PROGRAM MAIN
VAR
END_VAR

END_PROGRAM

(* stored: Version 1.1.0.1, ProductVersion 3.1.0.38
   POU MAIN: Id {00a7a124-c1e6-4562-adca-e98747e35c1e}, SpecialFunc None *)
